INTERFACE ITF_AnalogSensor

PROPERTY Value : INT
GET
END_GET
END_PROPERTY

END_INTERFACE

(* stored: Version 1.1.0.1
   Itf ITF_AnalogSensor: Id {06ce812f-1f4e-4e67-bebd-988fe75376d9}
   Property Value: Id {00f43883-91a0-486b-9268-9d7f1f7ae468}
   Get Get: Id {f866117e-a940-4646-a734-6253dc0153eb} *)
